FUNCTION_BLOCK FB_Manual_SC
VAR_INPUT
	bEnable			: BOOL;
	
END_VAR
VAR_OUTPUT
	fPCV				: LREAL;
	fSCV				: LREAL;
END_VAR
VAR
//Set fPCV
fPCV_set				: LREAL := 1.0;



//Function Blocks
fbDisplacementControl		: FB_DisplacementControl; //slik det er nå må Manuel SC være på for å endre dis, 
													  //kan endres til bare running og knappen

fbJoystick					: FB_Joystick;
fbGetStartPos				: FB_StartPos;
fbWinchVelIntegrator		: FB_Integrator;
fbPID_payloadpos			: FB_PID_Controller_posref;
fbDeadband					: FB_Deadband;
fbDisplacementControl_SC	: FB_DisplacementControl_SC;

fbMUX_selector				: FB_MUX_selector;

fbTarget_dis				: FB_Target_displacement;
fbGain_Chooser_P			: FB_GainChooser;
fbGain_Chooser_I			: FB_GainChooser;

//Variables
fWinchVelRefManual			: LREAL;
fWinchVelRefAuto			: LREAL;
fInitialWinchPos			: LREAL;

//Deaband
fUpperdeadband				: LREAL := 0.5;
fLowerdeadband				: LREAL := 0.14;
fNeutraldeadband			: LREAL := 0.35;
fDeadbandComp_out			: LREAL;

//Outer Loop output
fSC_ClosedLoopSingal		: LREAL;

//Valve signals
fSCV_target					: LREAL;
fSCV_Posref					: LREAL;
fSCV_Off					: LREAL;

fPCV_On						: LREAL;
fPCV_Off					: LREAL;

//DisplacementControl justering med slider på x akse ikke lagt til



END_VAR
VAR // added by the converter: edge detectors and wires of the graphical bodies
    _w1 : BOOL;
END_VAR

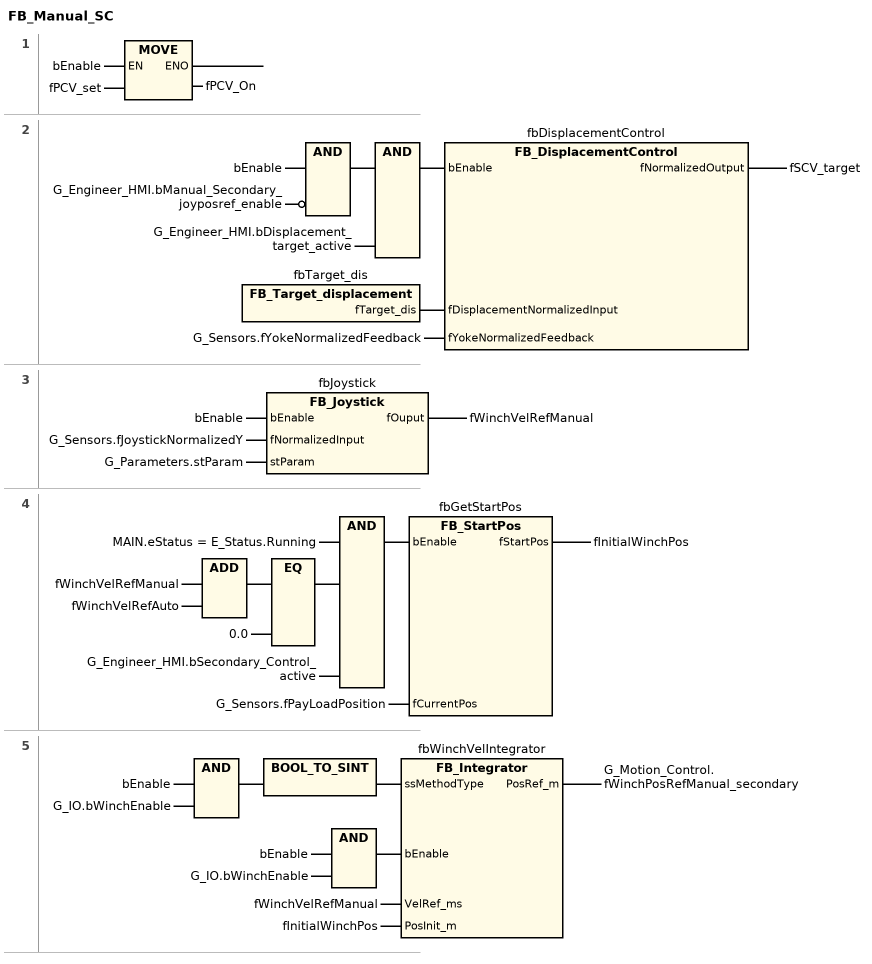
// NETWORK 1
IF bEnable THEN fPCV_On := fPCV_set; END_IF

// NETWORK 2
fbTarget_dis(); // FB_Target_displacement
fbDisplacementControl(
    bEnable := (bEnable AND NOT G_Engineer_HMI.bManual_Secondary_joyposref_enable) AND G_Engineer_HMI.bDisplacement_target_active,
    fDisplacementNormalizedInput := fbTarget_dis.fTarget_dis,
    fYokeNormalizedFeedback := G_Sensors.fYokeNormalizedFeedback); // FB_DisplacementControl
fSCV_target := fbDisplacementControl.fNormalizedOutput;

// NETWORK 3
fbJoystick(
    bEnable := bEnable,
    fNormalizedInput := G_Sensors.fJoystickNormalizedY,
    stParam := G_Parameters.stParam); // FB_Joystick
fWinchVelRefManual := fbJoystick.fOuput;

// NETWORK 4
fbGetStartPos(bEnable := (MAIN.eStatus = E_Status.Running) AND fWinchVelRefManual + fWinchVelRefAuto = 0.0 AND G_Engineer_HMI.bSecondary_Control_active, fCurrentPos := G_Sensors.fPayLoadPosition); // FB_StartPos
fInitialWinchPos := fbGetStartPos.fStartPos;

// NETWORK 5
fbWinchVelIntegrator(
    ssMethodType := BOOL_TO_SINT(bEnable AND G_IO.bWinchEnable),
    bEnable := bEnable AND G_IO.bWinchEnable,
    VelRef_ms := fWinchVelRefManual,
    PosInit_m := fInitialWinchPos); // FB_Integrator
G_Motion_Control.fWinchPosRefManual_secondary := fbWinchVelIntegrator.PosRef_m;

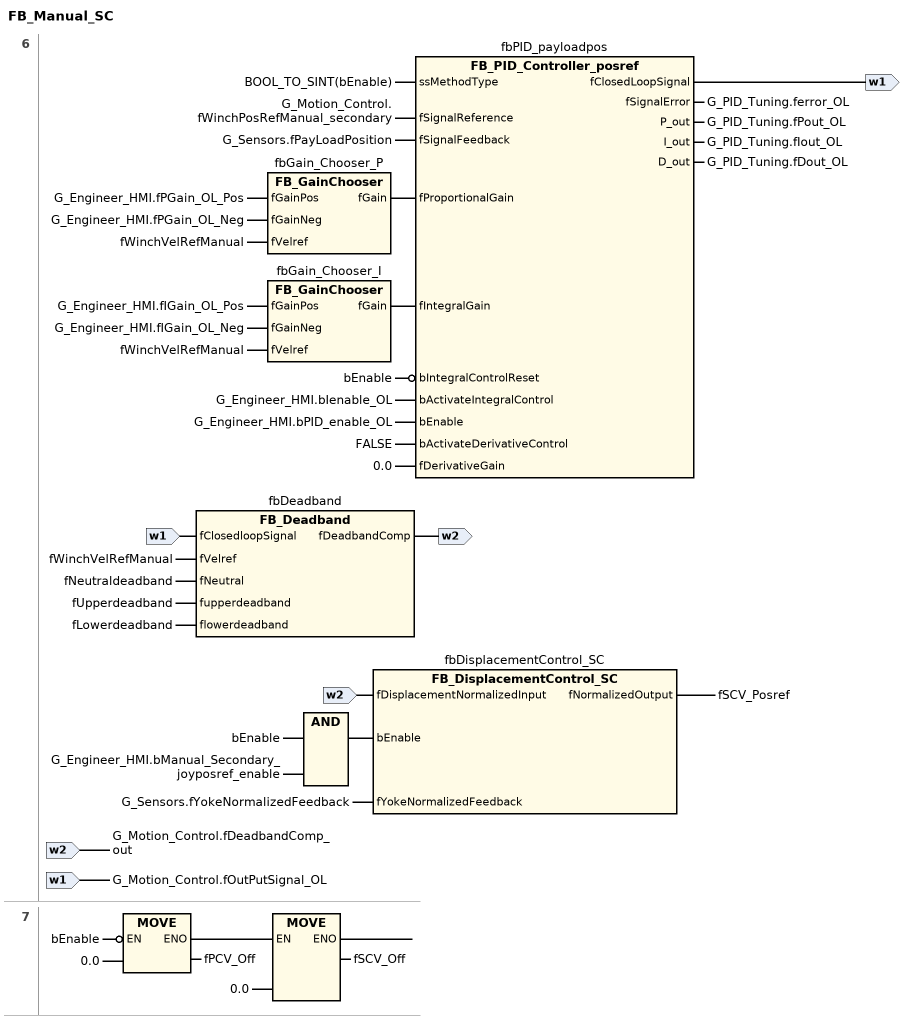
// NETWORK 6
fbGain_Chooser_P(
    fGainPos := G_Engineer_HMI.fPGain_OL_Pos,
    fGainNeg := G_Engineer_HMI.fPGain_OL_Neg,
    fVelref := fWinchVelRefManual); // FB_GainChooser
fbGain_Chooser_I(
    fGainPos := G_Engineer_HMI.fIGain_OL_Pos,
    fGainNeg := G_Engineer_HMI.fIGain_OL_Neg,
    fVelref := fWinchVelRefManual); // FB_GainChooser
fbPID_payloadpos(
    ssMethodType := BOOL_TO_SINT(bEnable),
    fSignalReference := G_Motion_Control.fWinchPosRefManual_secondary,
    fSignalFeedback := G_Sensors.fPayLoadPosition,
    fProportionalGain := fbGain_Chooser_P.fGain,
    fIntegralGain := fbGain_Chooser_I.fGain,
    bIntegralControlReset := NOT bEnable,
    bActivateIntegralControl := G_Engineer_HMI.bIenable_OL,
    bEnable := G_Engineer_HMI.bPID_enable_OL,
    bActivateDerivativeControl := FALSE,
    fDerivativeGain := 0.0,
    fSignalError => G_PID_Tuning.ferror_OL,
    P_out => G_PID_Tuning.fPout_OL,
    I_out => G_PID_Tuning.fIout_OL,
    D_out => G_PID_Tuning.fDout_OL); // FB_PID_Controller_posref
fbDeadband(
    fClosedloopSignal := fbPID_payloadpos.fClosedLoopSignal,
    fVelref := fWinchVelRefManual,
    fNeutral := fNeutraldeadband,
    fupperdeadband := fUpperdeadband,
    flowerdeadband := fLowerdeadband); // FB_Deadband
fbDisplacementControl_SC(
    fDisplacementNormalizedInput := fbDeadband.fDeadbandComp,
    bEnable := bEnable AND G_Engineer_HMI.bManual_Secondary_joyposref_enable,
    fYokeNormalizedFeedback := G_Sensors.fYokeNormalizedFeedback); // FB_DisplacementControl_SC
fSCV_Posref := fbDisplacementControl_SC.fNormalizedOutput;
G_Motion_Control.fDeadbandComp_out := fbDeadband.fDeadbandComp;
G_Motion_Control.fOutPutSignal_OL := fbPID_payloadpos.fClosedLoopSignal;

// NETWORK 7
_w1 := NOT bEnable;
IF _w1 THEN fPCV_Off := 0.0; END_IF
IF _w1 THEN fSCV_Off := 0.0; END_IF

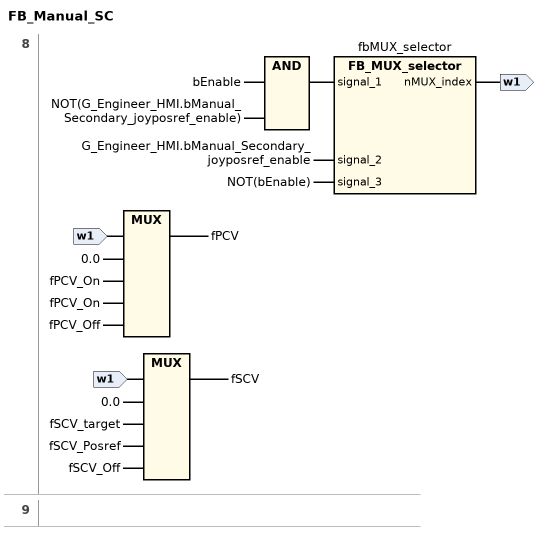
// NETWORK 8
fbMUX_selector(
    signal_1 := bEnable AND (NOT(G_Engineer_HMI.bManual_Secondary_joyposref_enable)),
    signal_2 := G_Engineer_HMI.bManual_Secondary_joyposref_enable,
    signal_3 := NOT(bEnable)); // FB_MUX_selector
fPCV := MUX(fbMUX_selector.nMUX_index, 0.0, fPCV_On, fPCV_On, fPCV_Off);
fSCV := MUX(fbMUX_selector.nMUX_index, 0.0, fSCV_target, fSCV_Posref, fSCV_Off);

// NETWORK 9

END_FUNCTION_BLOCK

(* stored: Version 1.1.0.1
   POU FB_Manual_SC: Id {9fac608f-03ce-4af0-a34b-044f392c42ef}, SpecialFunc None *)
